FUNCTION_BLOCK RequestOrchestrationForm (* Request Orchestration Function Block *)
  (* Standard: 61499-2; Description: Copyright (c) 2018 fortiss GmbH This program and the accompanying materials are made available under the terms of the Eclipse Public License 2.0 which is available at https://www.eclipse.org/legal/epl-2.0/ SPDX-License-Identifier: EPL-2.0 *)
  (* Version 1.0, 2018-09-21, Jose Cabral, fortiss GmbH *)
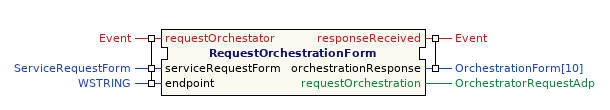
  EVENT_INPUT
    requestOrchestator WITH serviceRequestForm, endpoint; (* Request form to orchestrator *)
  END_EVENT
  EVENT_OUTPUT
    responseReceived WITH orchestrationResponse; (* A response was received from the orchestrator *)
  END_EVENT
  VAR_INPUT
    serviceRequestForm : ServiceRequestForm; (* Service request form to be sent to the orchestrator *)
    endpoint : WSTRING; (* Endpoint (IP:PORT/URI) of the orchestrator *)
  END_VAR
  VAR_OUTPUT
    orchestrationResponse : ARRAY [0..9] OF OrchestrationForm; (* Response from the orchestrator *)
  END_VAR
  PLUGS
    requestOrchestration : OrchestratorRequestAdp; (* Request Orchestration adapter *)
  END_PLUGS
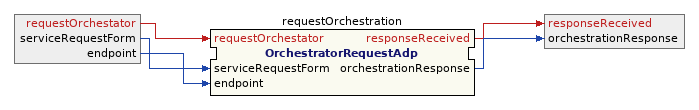
  EVENT_CONNECTIONS
    requestOrchestator TO requestOrchestration.requestOrchestator;
    requestOrchestration.responseReceived TO responseReceived;
  END_CONNECTIONS
  DATA_CONNECTIONS
    serviceRequestForm TO requestOrchestration.serviceRequestForm;
    requestOrchestration.orchestrationResponse TO orchestrationResponse;
    endpoint TO requestOrchestration.endpoint;
  END_CONNECTIONS
END_FUNCTION_BLOCK
